% RSLogix 500 project I2P JOB 7.RSS, saved by version 10.00.00.00 %
PROJECT "ML06B"    % processor: Bul.1763 MicroLogix 1100 Series B %

PROGRAM FILES
  LAD 2   5 rungs

DATA FILES
  O0 OUTPUT  4 elements
  I1 INPUT  6 elements
  S2 STATUS  66 elements
  B3 BINARY  1 elements
  T4 TIMER  1 elements
  C5 COUNTER  1 elements
  R6 CONTROL  1 elements
  N7 INTEGER  1 elements
  F8 FLOAT  1 elements

LADDER 2
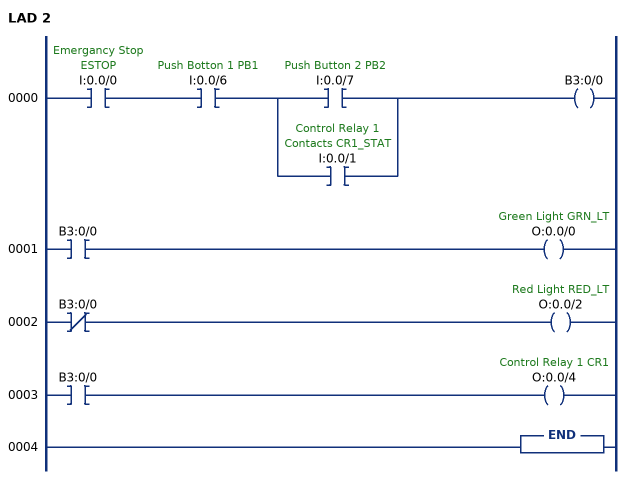
% Rung: 0 %
SOR XIC I:0.0/0 XIC I:0.0/6 BST XIC I:0.0/7 NXB XIC I:0.0/1 BND OTE B3:0/0 EOR
%   I:0.0/0  ESTOP  "Emergancy Stop" %
%   I:0.0/6  PB1  "Push Botton 1" %
%   I:0.0/7  PB2  "Push Button 2" %
%   I:0.0/1  CR1_STAT  "Control Relay 1 Contacts" %
% Rung: 1 %
SOR XIC B3:0/0 OTE O:0.0/0 EOR
%   O:0.0/0  GRN_LT  "Green Light" %
% Rung: 2 %
SOR XIO B3:0/0 OTE O:0.0/2 EOR
%   O:0.0/2  RED_LT  "Red Light" %
% Rung: 3 %
SOR XIC B3:0/0 OTE O:0.0/4 EOR
%   O:0.0/4  CR1  "Control Relay 1" %
% Rung: 4 %
SOR END EOR

OTHER DOCUMENTED ADDRESSES
  I:0.0/2  CR2_STAT  "Control Relay 2 Contacts"
  I:0.0/3  3PSS_A  "Three Position Selector Switch A Position"
  I:0.0/4  3PSS_B  "Three Postion Selector Switch B Position"
  I:0.0/5  2PSS_A  "Two Position Selector Switch A Position"
  I:0.0/8  PB3  "Push Botton 3"
  O:0.0/1  YLW_LT  "Yellow Light"
  O:0.0/3  BLU_LT  "Blue Light"
  O:0.0/5  CR2  "Control Relay 2"
